// TIA Portal V17 export
// export: Created 2024-09-02T12:50:25.2746861Z, ExportSetting WithDefaults, DisplayName Totally Integrated Automation Portal, DisplayVersion V17, DisplayName TIA Portal Openness, DisplayVersion V17, DisplayName TIA Portal Version Control Interface, DisplayVersion V17, DisplayName STEP 7 Professional, DisplayVersion V17, DisplayName STEP 7 Safety, DisplayVersion V17, DisplayName WinCC Professional, DisplayVersion V17
VAR_GLOBAL   // PLC tag table "VarAllgemein"
   QEKS_OP70 AT %Q7000.0 : "LTLL_typeEksInterface";   // EKS at the control panel / EKS am Bedienpult
   ibn0 AT %M10.0 : Bool;   // IBM flag with status 0 / IBM Merker mit Status 0
   ibn1 AT %M10.1 : Bool;   // IBM flag with status 1 / IBM Merker mit Status 1
   ibn_safety AT %M10.7 : Bool;   // IBM flag with status 1 for Safty / IBM Merker mit Status 1 für Safty
   dummy AT %M10.2 : Bool;   // Dummy flags / Dummymerker
   i_byte AT %I0.0 : "type_HW_Byte";   //    {ExternalAccessible false, ExternalVisible false, ExternalWritable false}
END_VAR
